Staubli VAL3: iSchock.pgx

public program iSchock(num& nNum[] (dimensions=1))
begin
  nNum=dioGet(iSchock)
end
